PROGRAM POU
VAR
	i	: LWORD;
END_VAR


RETURN;

i := i + 1;

END_PROGRAM

(* stored: Version 1.1.0.1
   POU POU: Id {d72a43ca-9f18-499f-9d7b-288c12cd0740}, SpecialFunc None *)
